SYSTEM SimultaneousEvents
  (* Version 1.0, 2005-12-22, Oscar, Chalmers *)
  DEVICE Test Device : DeviceType_not_used
    RESOURCE TestResource : ResourceType_not_used
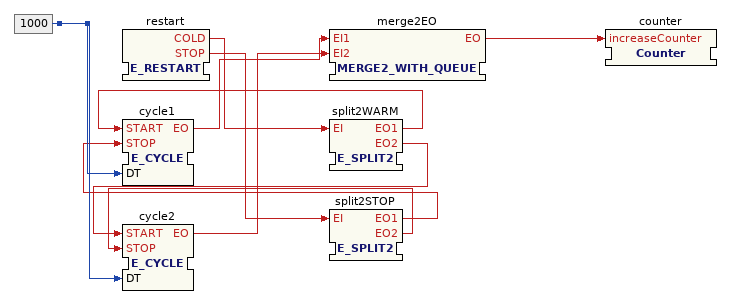
      FBS
        restart : E_RESTART;
        cycle1 : E_CYCLE;
        cycle2 : E_CYCLE;
        merge2EO : MERGE2_WITH_QUEUE;
        split2WARM : E_SPLIT2;
        split2STOP : E_SPLIT2;
        counter : Counter;
      END_FBS
      EVENT_CONNECTIONS
        restart.COLD TO split2WARM.EI;
        split2WARM.EO1 TO cycle1.START;
        split2WARM.EO2 TO cycle2.START;
        restart.STOP TO split2STOP.EI;
        split2STOP.EO1 TO cycle1.STOP;
        split2STOP.EO2 TO cycle2.STOP;
        cycle1.EO TO merge2EO.EI1;
        cycle2.EO TO merge2EO.EI2;
        cycle1.EO TO merge2EO.EI1;
        merge2EO.EO TO counter.increaseCounter;
      END_CONNECTIONS
      DATA_CONNECTIONS
        1000 TO cycle1.DT;
        1000 TO cycle2.DT;
      END_CONNECTIONS
    END_RESOURCE
  END_DEVICE
END_SYSTEM
(* other elements stored in the file *)
(* FB Name="delay" Type="E_DELAY" / *)
(* FB Name="merge2EO" Type="E_MERGE2" / *)
(* Connection Source="cycle2.EO" Destination="delay.START" / *)
(* Connection Source="delay.EO" Destination="merge2EO.EI2" / *)
(* Connection Source="1" Destination="delay.DT" / *)
